{attribute 'linkalways'} 
{attribute 'no_explicit_call' := 'This FB is a CLASS and must be accessed using methods or properties'}
{attribute 'enable_dynamic_creation'}
FUNCTION_BLOCK Node_F_VN_DetectCodesNeuralNetwork EXTENDS VisionNode
VAR
    ipSrcImage : _ITcVnImage;
    ipCodeRegions : _ITcVnContainer;
    ipCodeTypes : _ITcVnContainer;
	eModelType : _ETcVnCodeDetectionModel(ETcVnCodeDetectionModel.TCVN_CDM_DETECT_1_1);
	nCodeType : _ULINT(0);
    hrPrev : _HRESULT(S_OK);
	hresult : _HRESULT(S_OK);
END_VAR

METHOD PUBLIC  Clone : I_Node
VAR
	pNode : POINTER TO Node_F_VN_DetectCodesNeuralNetwork;
END_VAR
pNode := __NEW(Node_F_VN_DetectCodesNeuralNetwork);
Clone := pNode^;
END_METHOD

METHOD FB_init : BOOL
VAR_INPUT
	bInitRetains : BOOL; // if TRUE, the retain variables are initialized (warm start / cold start)
	bInCopyCode : BOOL;  // if TRUE, the instance afterwards gets moved into the copy code (online change)
END_VAR
AddInput('ipSrcImage', ipSrcImage);
AddInput('eModelType', eModelType);
AddInput('nCodeType', nCodeType);
AddInput('hrPrev', hrPrev);
AddOutput('ipCodeRegions', ipCodeRegions);
AddOutput('ipCodeTypes', ipCodeTypes);
AddOutput('hresult', hresult);
END_METHOD

METHOD PROTECTED OnExecute
hresult.Value := F_VN_DetectCodesNeuralNetwork(
	ipSrcImage := ipSrcImage.Value,
	ipCodeRegions := ipCodeRegions.Value,
	ipCodeTypes := ipCodeTypes.Value,
    eModelType := eModelType.Value,
    nCodeType := nCodeType.Value,
	hrPrev:= hrPrev.Value
);
END_METHOD

METHOD PUBLIC PreExecutionCheck
VAR_INPUT
	Check : I_PreExecutionChecks;
END_VAR
Check.IsTrue(ipSrcImage.IsValid, 'ipSrcImage must contain an image');
Check.IsTrue((ipSrcImage.HasChannelCount(1) OR ipSrcImage.HasChannelCount(3)), 'ipSrcImage must contain 1 or 3 channels');
END_METHOD

END_FUNCTION_BLOCK

(* stored: Version 1.1.0.1, ProductVersion 3.1.4026.13
   POU Node_F_VN_DetectCodesNeuralNetwork: Id {2954f261-37ad-044e-1502-8517de237731}, SpecialFunc None
   Folder Constructor: Id {9877e2b4-a773-081a-32b2-0882bc63ba44}
   Method Clone: Id {7aba535b-c048-097d-0fd9-d379d59eeebc}
   Method FB_init: Id {63bc7530-2eac-0c6e-09eb-54d02e6e4f3e}
   Method OnExecute: Id {8a7fe928-13c8-009f-2ab3-c04ce677c044}
   Method PreExecutionCheck: Id {b147fdef-7073-00da-271d-277637ca66a3} *)
